// TwinCAT 3 PLC project B3TrafficLight_Plc
// Title: B3TrafficLight_Plc
// Company: Tc3 Project
// ProjectVersion: 1.0.0.0
// ProgramVersion: 3.1.4026.22
// libraries:
//   Tc2_Standard, * (Beckhoff Automation GmbH)
//   Tc2_System, * (Beckhoff Automation GmbH)
// project tree:
//   / PlcTask.TcTTO
//   POUs/ FB_TrafficLight.TcPOU, MAIN.TcPOU
// real-time tasks:
//   TASK PlcTask: cycle T#10ms, priority 20, ADS port 350

CONFIGURATION B3TrafficLight_Plc
    RESOURCE PLC ON TwinCAT3
        TASK PlcTask(INTERVAL := T#10ms, PRIORITY := 20);
        PROGRAM MAIN WITH PlcTask : MAIN;
    END_RESOURCE
END_CONFIGURATION

// ---- POUs/MAIN.TcPOU
PROGRAM MAIN
VAR
END_VAR

END_PROGRAM

// ---- POUs/FB_TrafficLight.TcPOU
FUNCTION_BLOCK FB_TrafficLight
VAR
    state : INT;  // 0=Red, 1=RedAmber, 2=Green, 3=Amber
END_VAR

METHOD Step : INT
CASE state OF
    0:
        state := 1;
    1:
        state := 2;
    2:
        state := 0;
    3:
        state := 0;
END_CASE;
Step := state;
END_METHOD

END_FUNCTION_BLOCK
